{region '#Template'}
	{attribute 'Version' := '5.0.1.0'}
	{attribute 'Tags' := '"LCID": "1031", "Text": "H, Plant, HtgCir, Heating circuit"'}
	{attribute 'Tags' := '"LCID": "1033", "Text": "H, Plant, HtgCir, Heating circuit"'}
	{attribute 'Using' := '"Type": "Template", "URI": "Site"'}
	{attribute 'Description' := '"LCID": "1031", "Text": "Heizkreis"'}
	{attribute 'Description' := '"LCID": "1033", "Text": "Heating circuit"'}
{endregion}
FUNCTION_BLOCK FB_BA_H_HtgCir01 EXTENDS FB_BA_View
VAR_INPUT
END_VAR
VAR_OUTPUT
	eOpMod 					: E_BA_EnergyLvl;
	bRls					: BOOL;	
	fSp    					: REAL;
	bPu    					: BOOL;
	fVlv   					: REAL;
END_VAR
VAR_INPUT CONSTANT
	TFl						: FB_BA_SensorAnalog;												
	TRt						: FB_BA_SensorAnalog;																									
	Vlv						: FB_BA_Vlv;									
	Pu						: FB_BA_Pu1st;	
	Sp						: FB_BA_H_HtgCir_Sp;												
	OpMod					: FB_BA_H_OpMod;									
	HtgLmt					: FB_BA_HtgLmt;							
	TFlCtrl					: FB_BA_PID;
	PlantLock				: FB_BA_PlantLock;	
END_VAR
VAR
END_VAR
VAR // added by the converter: edge detectors and wires of the graphical bodies
    _s1 : ST_BA_Analog;
    _s2 : ST_BA_Binary;
    _w1 : ANY;
END_VAR

// note: 14 stored wires end on pins the file does not list and are not shown
SUPER^(); // FB_BA_View
TFl(); // FB_BA_SensorAnalog
TRt(); // FB_BA_SensorAnalog
PlantLock(); // FB_BA_PlantLock
_w1 := PlantLock.bPrioHigh OR PlantLock.bPrioMedium;
HtgLmt(fIn := Site.stGeneralSettings.fTWthDamped); // FB_BA_HtgLmt
OpMod(bDst := _w1, bHtgLmt := HtgLmt.bQ, bTWthLowLimit := Site.stGeneralSettings.bTWthLowLimit); // FB_BA_H_OpMod
bRls := OpMod.bRls;
eOpMod := OpMod.eOpMod;
Sp(
    eOpMod := eOpMod,
    fSpFrstProtec := Site.stGeneralSettings.fFrostProtectionSetpoint,
    fTWthDamp := Site.stGeneralSettings.fTWthDamped); // FB_BA_H_HtgCir_Sp
fSp := Sp.fSpFlWT;
TFlCtrl(bEn := OpMod.bRls, fW := fSp, fX := TFl.fPresentValue); // FB_BA_PID
// compose _s1 : ST_BA_Analog
_s1.bEnSfty := PlantLock.bPrioHigh;
_s1.fValSfty := 0;
_s1.bEnCrit := PlantLock.bPrioMedium;
_s1.fValCrit := 0;
_s1.bEnPgm := OpMod.bRls;
_s1.fValPgm := TFlCtrl.fY;
// compose _s2 : ST_BA_Binary
_s2.bEnSfty := PlantLock.bPrioHigh;
_s2.bValSfty := FALSE;
_s2.bEnCrit := PlantLock.bPrioMedium;
_s2.bValCrit := FALSE;
_s2.bEnPgm := OpMod.bRls;
_s2.bValPgm := TRUE;
Pu(stCmd := _s2, bAblkLock := fVlv >= 10.0); // FB_BA_Pu1st
bPu := Pu.bCmd;
Vlv(stCmd := _s1, bAblkLock := Pu.bCmd); // FB_BA_Vlv
fVlv := Vlv.fMdlt;

METHOD FB_init : BOOL
VAR_INPUT
	bInitRetains : BOOL; // if TRUE, the retain variables are initialized (warm start / cold start)
	bInCopyCode : BOOL;  // if TRUE, the instance afterwards gets moved into the copy code (online change)
END_VAR
PlantLock.Parent						:= THIS^;		

TFl.iParent								:= THIS^;	
TFl.iLabel								:= LblAgg_TemperatureFlow; 
TFl.eDPADMode							:= E_BA_DPADMode.eInclude;																																	
TFl.MV.eUnit							:= E_BA_Unit.eTemperature_DegreesCelsius;
TFl.MV.fResolution 						:= 0.01;
TFl.MV.fScaleOffset 					:= 0; 
TFl.MV.bEventDetectionEnable			:= TRUE;
TFl.MV.eEnPlantLock						:= E_BA_LockPriority.eMedium;

TRt.iParent								:= THIS^;		
TRt.iLabel								:= LblAgg_TemperatureReturnFlow; 
TRt.eDPADMode							:= E_BA_DPADMode.eInclude;																																	
TRt.MV.eUnit							:= E_BA_Unit.eTemperature_DegreesCelsius;
TRt.MV.fResolution 						:= 0.01;
TRt.MV.fScaleOffset 					:= 0;  
TRt.MV.bEventDetectionEnable			:= TRUE;
TRt.MV.eEnPlantLock						:= E_BA_LockPriority.eNoLock;
				
Vlv.iParent								:= THIS^;	
Vlv.iLabel								:= LblAgg_Valve; 
Vlv.eDPADMode							:= E_BA_DPADMode.eInclude;									
				
Pu.iParent								:= THIS^;
Pu.iLabel								:= LblAgg_Pump; 
Pu.eDPADMode							:= E_BA_DPADMode.eInclude;	
Pu.Dst.bEventDetectionEnable			:= TRUE;			
				
Sp.iParent								:= THIS^;	
Sp.iLabel								:= LblCtl_SetpointGeneration; 
Sp.eDPADMode							:= E_BA_DPADMode.eInclude;												
				
OpMod.iParent							:= THIS^;	
OpMod.iLabel							:= LblCtl_OperationMode; 
OpMod.eDPADMode							:= E_BA_DPADMode.eInclude;									
				
HtgLmt.iParent							:= THIS^;	
HtgLmt.iLabel							:= LblCtl_HeatingLimit; 
HtgLmt.eDPADMode						:= E_BA_DPADMode.eInclude;

TFlCtrl.iParent							:= THIS^;
TFlCtrl.iLabel							:= LblCtl_FlowTemperatureControl; 
TFlCtrl.eDPADMode						:= E_BA_DPADMode.eInclude;																																	
TFlCtrl.Ctrl.eOutputUnit				:= E_BA_Unit.eOther_Percent;
TFlCtrl.Ctrl.eActionRm					:= E_BA_Action.eReverse;
TFlCtrl.Ctrl.fMinOutputRm				:= 0;
TFlCtrl.Ctrl.fMaxOutputRm				:= 100;
TFlCtrl.Ctrl.fProportionalConstant		:= 3;
TFlCtrl.Ctrl.fIntegralConstant			:= 180;
END_METHOD

END_FUNCTION_BLOCK

(* stored: Version 1.1.0.1, ProductVersion 3.1.4024.12
   POU FB_BA_H_HtgCir01: Id {91ddc094-0dad-4f94-b06b-e7c6d99acc73}, SpecialFunc None
   Method FB_init: Id {316fd3be-1bf1-4183-b0e0-0cd1012c472a} *)
